FUNCTION_BLOCK FB_StairwellLight IMPLEMENTS ILight
VAR
	bControlValue		: BOOL;
	fbTon				: TON := (PT := TIME#3s0ms);
END_VAR

METHOD M_Execution
fbTon();
IF (fbTon.Q) THEN
	THIS^.M_Off();
END_IF
END_METHOD

PROPERTY P_ControlValue : BOOL
GET
P_ControlValue := bControlValue;
END_GET
SET
bControlValue := P_ControlValue;
END_SET
END_PROPERTY

METHOD M_On
P_ControlValue := TRUE;
fbTon(IN := TRUE);
END_METHOD

METHOD M_Off
P_ControlValue := FALSE;
fbTon(IN := FALSE);
END_METHOD

END_FUNCTION_BLOCK

(* stored: Version 1.1.0.1, ProductVersion 3.1.0.23
   POU FB_StairwellLight: Id {79c55de8-ccf9-4597-abb4-0bbb5aa395ab}
   Method M_Execution: Id {35a4aad4-009e-4f1a-9112-614c2c4d4b18}
   Property P_ControlValue: Id {6a2201ed-d1dd-438a-9303-4922b0bf3678}
   Get Get: Id {0e696bef-4d2a-43ac-a71d-38b653a521cd}
   Set Set: Id {57dd2b86-ea29-494d-8e8c-9c624dae1cae}
   Method M_On: Id {c5f9a38b-ceb1-4d0e-952a-1d697d4a5ea5}
   Method M_Off: Id {fbe6cfee-642c-4e29-b0bd-1767ede94dcb} *)
